FUNCTION_BLOCK MotionFunc

VAR CONSTANT
	AXIS_MIN_IDX : USINT := 1;
	AXIS_MAX_IDX : USINT := 6;
END_VAR

VAR_IN_OUT
	Axes : ARRAY[AXIS_MIN_IDX..AXIS_MAX_IDX] OF AXIS_REF;
	
END_VAR

VAR_INPUT
	Execute : BOOL;
	Mode : E_6Axis_Motion;
	StartPosition : ARRAY [1..6] OF LREAL;
	FinalPosition : ARRAY [1..6] OF LREAL;
	UpdateTime : LREAL;
END_VAR

VAR_OUTPUT
	Done : BOOL;
END_VAR

VAR
	idx : DINT;
	timer : LREAL;
	lastExecute : BOOL;
	six_pos : ARRAY [1..6, 1..6] OF LREAL;
	
	AbsMove : ARRAY [AXIS_MIN_IDX..AXIS_MAX_IDX] OF MC_MoveAbsolute;
	ExtSwitchEn : ARRAY [AXIS_MIN_IDX..AXIS_MAX_IDX] OF MC_ExtSetPointGenEnable;
	ExtSwitchDis : ARRAY [AXIS_MIN_IDX..AXIS_MAX_IDX] OF MC_ExtSetPointGenDisable;

	// PTP
	ptp_angles : ARRAY[1..6] OF LREAL;
 
	// linear
	pos : LREAL;
	vel : LREAL;
	acc : LREAL;
	direction : DINT;
	MF : MathFunc;
	KM : Kinematics;
	RunTimeCopy : LREAL;
	CoeffCopy : ARRAY[1..6, 1..6] OF LREAL; 
	UpdateTimeCopy : LREAL;
	
END_VAR

IF NOT Execute THEN
	Done := FALSE;
	lastExecute := Execute;
	RETURN;
END_IF

IF NOT lastExecute THEN
	CASE Mode OF 
		E_6Axis_Motion.PTP:
			mode_PTP(StartPosition, FinalPosition, angles => ptp_angles);
			FOR idx := AXIS_MIN_IDX TO AXIS_MAX_IDX DO
				AbsMove[idx].Execute := TRUE;
			END_FOR
			
			
		E_6Axis_Motion.LINEAR:
			MF.FindForSixPoints(StartPosition, FinalPosition, six_pos => six_pos);
			mode_Linear(six_pos, full_time => RunTimeCopy, coeffCopy => CoeffCopy);
			updateTimeCopy := UpdateTime;
			timer := 0;
	END_CASE
END_IF

lastExecute := Execute;



IF NOT Done THEN
	timer := timer + updateTimeCopy;
END_IF

Update_Absolute_Motion();
Update_Custom_Motion();
ActCustomMove();

ACTION ActCustomMove:
FOR idx := 1 TO 6 DO
	CASE Mode OF
		E_6Axis_Motion.PTP:
			AbsMove[idx].Position := ptp_angles[idx];
			AbsMove[idx].Velocity := 500;
		
		E_6Axis_Motion.Linear:
			pos := CoeffCopy[idx, 1]*EXPT(timer, 5) + CoeffCopy[idx, 2]*EXPT(timer, 4)	
				+ CoeffCopy[idx, 3]*EXPT(timer, 3) + CoeffCopy[idx, 4]*EXPT(timer, 2) 
				+ CoeffCopy[idx, 5]*EXPT(timer, 1) + CoeffCopy[idx, 6]*EXPT(timer, 0);
										  
			vel := CoeffCopy[idx, 1]*5*EXPT(timer, 4) + CoeffCopy[idx, 2]*4*EXPT(timer, 3)
				+ CoeffCopy[idx, 3]*3*EXPT(timer, 2) + CoeffCopy[idx, 4]*2*EXPT(timer, 1)
				+ CoeffCopy[idx, 5]*1*EXPT(timer, 0);
				 
			acc := CoeffCopy[idx, 1]*20*EXPT(timer, 3) + CoeffCopy[idx, 2]*12*EXPT(timer, 2)
				+ CoeffCopy[idx, 3]*6*EXPT(timer, 1) + CoeffCopy[idx, 4]*2*EXPT(timer, 0);
				
			IF vel = 0 AND acc = 0 THEN
				direction := 0;	(* stand still *)
			ELSIF vel >= 0 THEN
				direction := 1;	(* positive motion *)
			ELSE
				direction := -1;  (* negative motion *)
			END_IF
			
			IF timer >= runTimeCopy THEN
				vel := 0;
				acc := 0;
				direction := 0;
				Done := TRUE;
			END_IF
					
			MC_ExtSetPointGenFeed(
				Position := pos,
				Velocity := vel,
				Acceleration := acc,
				Direction := direction,
				Axis := Axes[idx]);	
				
	END_CASE
END_FOR
END_ACTION

METHOD mode_Linear : BOOL

VAR_INPUT
	six_pos : ARRAY [1..6, 1..6] OF LREAL;
END_VAR

VAR_OUTPUT
	full_time : LREAL;
	coeffCopy : ARRAY [1..6, 1..6] OF LREAL;
END_VAR

VAR
	idx : DINT;
	i, j : DINT;
	temp : LREAL; // 導正係數用

	pos01, pos02 : ARRAY [1..6] OF LREAL; //start and final point
	temp_pos : ARRAY [1..6] OF LREAL;
	temp_ang : ARRAY [1..6] OF LREAL;
	six_pos_angles : ARRAY [1..6, 1..6] OF LREAL;
	
	longest_distance : LREAL;
	time_factor : LREAL;
	
	six_time : ARRAY [1..6, 1..6] OF LREAL;
	timeCopy : ARRAY [1..6, 1..6] OF LREAL;
	
END_VAR
// Angles_mat
FOR i := 1 TO 6 DO
	FOR j := 1 TO 6 DO
		temp_pos[j] := six_pos[i, j];
	END_FOR
	KM.Inverse(position := temp_pos, angles => temp_ang);
	FOR j := 1 TO 6 DO
		six_pos_angles[j, i] := temp_ang[j];
	END_FOR
END_FOR

FOR idx := 1 TO 6 DO
	pos01[idx] := six_pos[1, idx];
	pos02[idx] := six_pos[6, idx];
END_FOR
longest_distance := SQRT(EXPT(pos02[1] - pos01[1], 2) + EXPT(pos02[2] - pos01[2], 2) + EXPT(pos02[3] - pos01[3], 2));
time_factor := EXPT(30, -1); // The larger the denominator, the faster the speed
full_time := time_factor * longest_distance;
//fix time proble
full_time := LREAL_TO_DINT(full_time * 1000)/1000;

// time_mat
FOR i := 1 TO 6 DO
	six_time[1, i] := 1;
	six_time[2, i] := (full_time)/5 * (i-1);
	FOR j := 3 TO 6 DO
		six_time[j, i] := EXPT(six_time[2, i], j-1);
	END_FOR
END_FOR

FOR i := 1 TO 6 DO
	FOR j := 1 TO 6 DO
		coeffCopy[i, j] := 0; // clear temp
		timeCopy[i, j] := six_time[i, j];
	END_FOR
END_FOR

MF.GaussianElimination(base_mat := timeCopy, extend_mat := six_pos_angles, temp_mat := coeffCopy, 6); //inverse 會搞壞原本的東西

FOR i := 1 TO 6 DO
	FOR j := 1 TO 3 DO
		temp := coeffCopy[i, j];
		coeffCopy[i, j] := coeffCopy[i, 7-j];
		coeffCopy[i, 7-j] := temp;
	END_FOR		
END_FOR
END_METHOD

METHOD mode_PTP : BOOL

VAR_INPUT
	start_pos : ARRAY [1..6] OF LREAL;
	final_pos : ARRAY [1..6] OF LREAL;
END_VAR

VAR_OUTPUT
	angles : ARRAY[1..6] OF LREAL; 
END_VAR

VAR
	
END_VAR
KM.Inverse(position := final_pos, angles => angles);
END_METHOD

ACTION Update_Absolute_Motion:
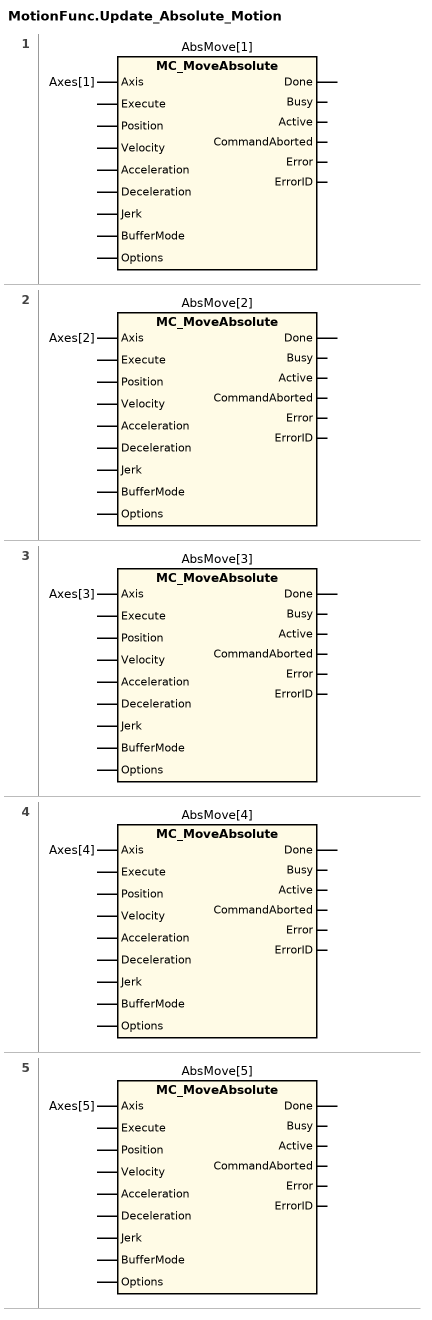
// NETWORK 1
AbsMove[1](Axis := Axes[1]); // MC_MoveAbsolute

// NETWORK 2
AbsMove[2](Axis := Axes[2]); // MC_MoveAbsolute

// NETWORK 3
AbsMove[3](Axis := Axes[3]); // MC_MoveAbsolute

// NETWORK 4
AbsMove[4](Axis := Axes[4]); // MC_MoveAbsolute

// NETWORK 5
AbsMove[5](Axis := Axes[5]); // MC_MoveAbsolute

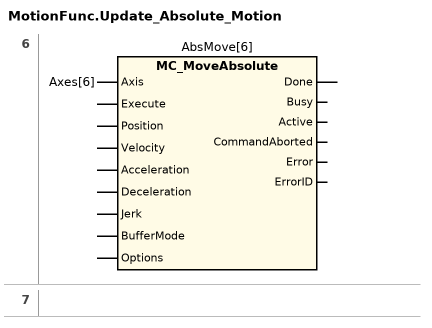
// NETWORK 6
AbsMove[6](Axis := Axes[6]); // MC_MoveAbsolute

// NETWORK 7
END_ACTION

ACTION Update_Custom_Motion:
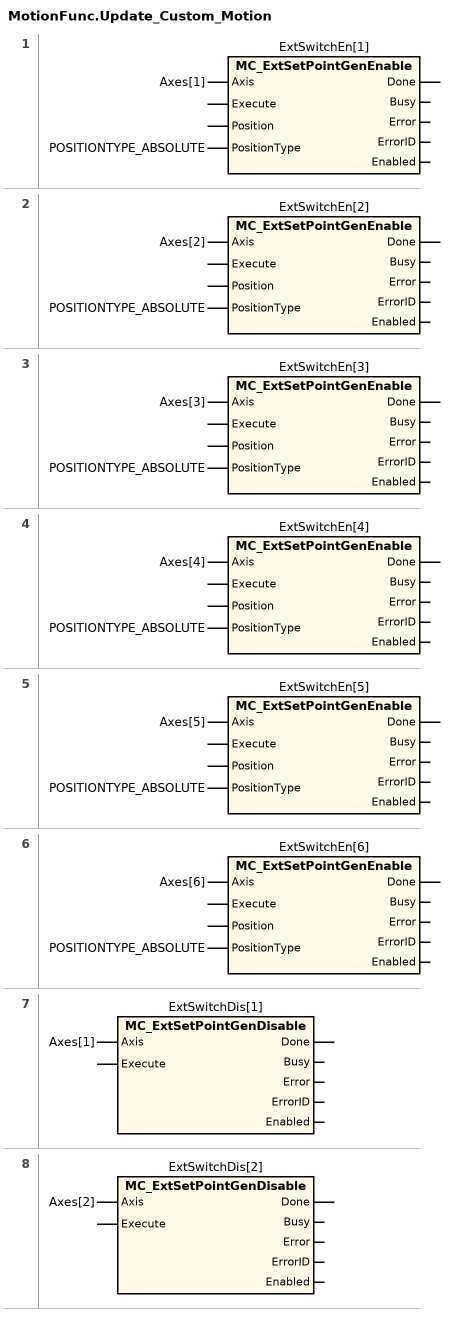
// NETWORK 1
ExtSwitchEn[1](Axis := Axes[1], PositionType := POSITIONTYPE_ABSOLUTE); // MC_ExtSetPointGenEnable

// NETWORK 2
ExtSwitchEn[2](Axis := Axes[2], PositionType := POSITIONTYPE_ABSOLUTE); // MC_ExtSetPointGenEnable

// NETWORK 3
ExtSwitchEn[3](Axis := Axes[3], PositionType := POSITIONTYPE_ABSOLUTE); // MC_ExtSetPointGenEnable

// NETWORK 4
ExtSwitchEn[4](Axis := Axes[4], PositionType := POSITIONTYPE_ABSOLUTE); // MC_ExtSetPointGenEnable

// NETWORK 5
ExtSwitchEn[5](Axis := Axes[5], PositionType := POSITIONTYPE_ABSOLUTE); // MC_ExtSetPointGenEnable

// NETWORK 6
ExtSwitchEn[6](Axis := Axes[6], PositionType := POSITIONTYPE_ABSOLUTE); // MC_ExtSetPointGenEnable

// NETWORK 7
ExtSwitchDis[1](Axis := Axes[1]); // MC_ExtSetPointGenDisable

// NETWORK 8
ExtSwitchDis[2](Axis := Axes[2]); // MC_ExtSetPointGenDisable

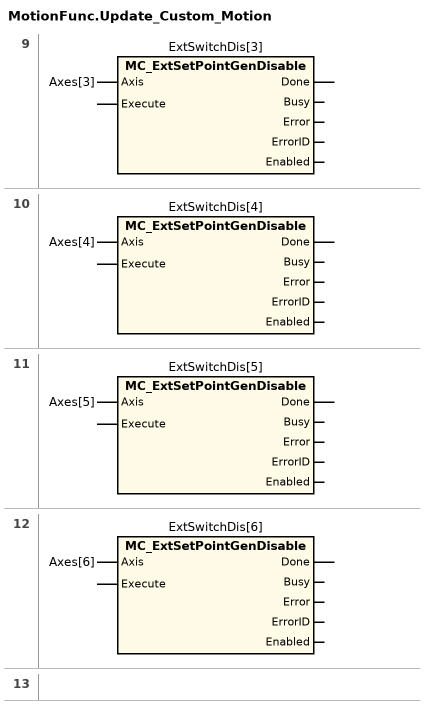
// NETWORK 9
ExtSwitchDis[3](Axis := Axes[3]); // MC_ExtSetPointGenDisable

// NETWORK 10
ExtSwitchDis[4](Axis := Axes[4]); // MC_ExtSetPointGenDisable

// NETWORK 11
ExtSwitchDis[5](Axis := Axes[5]); // MC_ExtSetPointGenDisable

// NETWORK 12
ExtSwitchDis[6](Axis := Axes[6]); // MC_ExtSetPointGenDisable

// NETWORK 13
END_ACTION

END_FUNCTION_BLOCK

(* stored: Version 1.1.0.1, ProductVersion 3.1.4024.12
   POU MotionFunc: Id {5c9f337a-07bb-402c-822f-794d1f4cbf9c}, SpecialFunc None
   Action ActCustomMove: Id {d2dff6a7-40fb-40d5-8d99-77f853e148b3}
   Method mode_Linear: Id {daa39aef-e9f0-4f2c-b084-defdf4f5c29b}
   Method mode_PTP: Id {dece690c-5394-4d47-96e3-4545268fd10c}
   Action Update_Absolute_Motion: Id {98d5d950-8383-448d-a5fb-12c28acbf0e2}
   Action Update_Custom_Motion: Id {52e3c804-ad23-48a4-b377-f256b01cdf0b} *)
